# EPICS autosave request: ipApp/Db/ADAM_4018_chan_settings.req
$(P)$(R):ai$(C).DESC
$(P)$(R):temp$(C).DESC
$(P)$(R):unit$(C).VAL
